// Mitsubishi GX Works2 project: inverter2   PLC: Q03UDV

PROGRAM MAIN
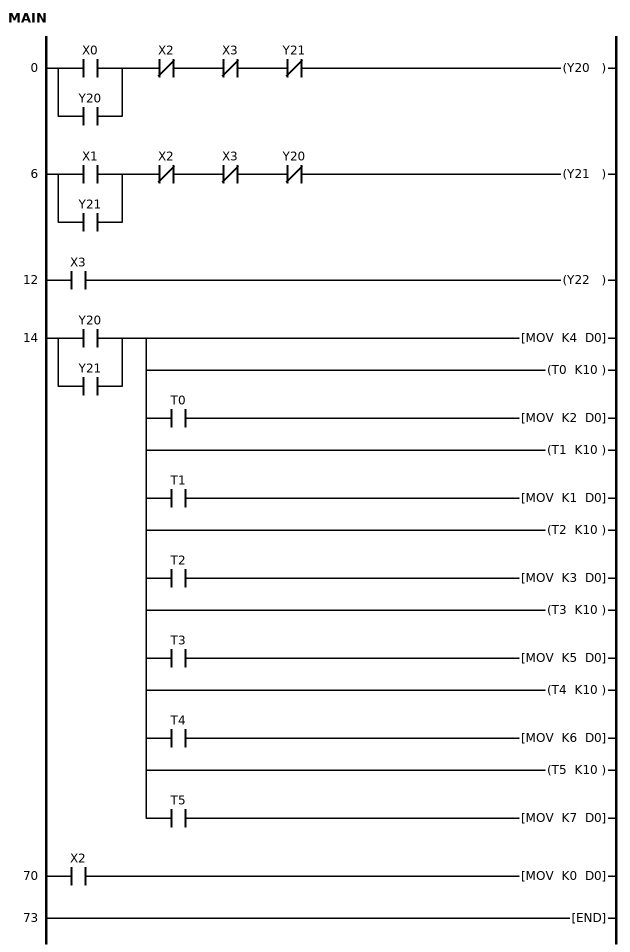
0     LD      X0
      OR      Y20
      ANI     X2
      ANI     X3
      ANI     Y21
      OUT     Y20
6     LD      X1
      OR      Y21
      ANI     X2
      ANI     X3
      ANI     Y20
      OUT     Y21
12    LD      X3
      OUT     Y22
14    LD      Y20
      OR      Y21
      MOV     K4 D0
      OUT     T0 K10
      MPS
      AND     T0
      MOV     K2 D0
      MPP
      OUT     T1 K10
      MPS
      AND     T1
      MOV     K1 D0
      MPP
      OUT     T2 K10
      MPS
      AND     T2
      MOV     K3 D0
      MPP
      OUT     T3 K10
      MPS
      AND     T3
      MOV     K5 D0
      MPP
      OUT     T4 K10
      MPS
      AND     T4
      MOV     K6 D0
      MPP
      OUT     T5 K10
      AND     T5
      MOV     K7 D0
70    LD      X2
      MOV     K0 D0
73    END
END_PROGRAM

PROGRAM MAIN1
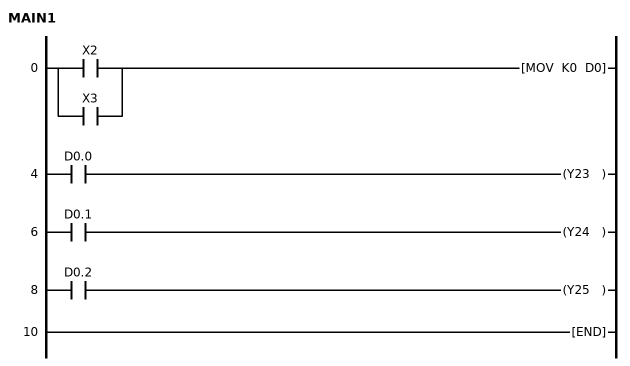
0     LD      X2
      OR      X3
      MOV     K0 D0
4     LD      D0.0
      OUT     Y23
6     LD      D0.1
      OUT     Y24
8     LD      D0.2
      OUT     Y25
10    END
END_PROGRAM
